// Mitsubishi GX Works2 project: GX W2 L5 Ex 3 DK C   PLC: FX3G

// task Task_01 (event TRUE, interval 0, priority 31): POU_01

PROGRAM POU_01
VAR
  wWallStat : INT;
  bHeater : BOOL;
END_VAR
IF wWallStat < 18 THEN
	bHeater := 1;
ELSE
	bHeater := 0;
END_IF;
END_PROGRAM
